// TwinCAT 3 PLC project program1
// ProgramVersion: 3.1.4023.0
// libraries:
//   Tc2_Standard, * (Beckhoff Automation GmbH)
//   Tc2_System, * (Beckhoff Automation GmbH)
//   Tc3_Module, * (Beckhoff Automation GmbH)
// project tree:
//   GVLs/ Common_GVL.TcGVL, ST_Siemens_data_inputs.TcDUT, ST_Siemens_data_outputs.TcDUT, ST_Siemens_other_parameters.TcDUT, ST_Siemens_production_data.TcDUT
//   / PlcTask.TcTTO
//   POUs/ FB_TestFunction.TcPOU, MAIN.TcPOU
// real-time tasks:
//   TASK PlcTask: cycle T#10ms, priority 20, ADS port 350
//   TASK Device 1 (OPC UA Virtual)_Task_58: cycle T#40ms, priority 58, ADS port 351
// I/O:
//   DEVICE Device 1 (OPC UA Virtual), AmsNetId 192.168.0.5.2.1
// variable links:
//   program1/program1 Instance <-> Device 1 (OPC UA Virtual)/Client #1/ServerInterfaces.Communication_with_beckhoff.Bottle_Count
//     PlcTask Inputs/TestData.xBottleCount <-> Inputs/Value
//   program1/program1 Instance <-> Device 1 (OPC UA Virtual)/Client #1/ServerInterfaces.Communication_with_beckhoff.Flow_ml_per_sec
//     PlcTask Inputs/TestData.rFlow_in_ml_s <-> Inputs/Value
//   program1/program1 Instance <-> Device 1 (OPC UA Virtual)/Client #1/ServerInterfaces.Communication_with_beckhoff.LiquidA_in_Bottle
//     PlcTask Inputs/TestData.aryLiquidA_in_bottle <-> Inputs/Value
//     PlcTask Inputs/TestData.aryLiquidA_in_bottle[{0..5}] <-> Inputs/Value[{0..5}]  (6 links)
//   program1/program1 Instance <-> Device 1 (OPC UA Virtual)/Client #1/ServerInterfaces.Communication_with_beckhoff.LiquidB_in_Bottle
//     PlcTask Inputs/TestData.aryLiquidB_in_bottle <-> Inputs/Value
//     PlcTask Inputs/TestData.aryLiquidB_in_bottle[{0..5}] <-> Inputs/Value[{0..5}]  (6 links)
//   program1/program1 Instance <-> Device 1 (OPC UA Virtual)/Client #1/ServerInterfaces.Communication_with_beckhoff.T02_Level_in_L
//     PlcTask Inputs/TestData.rT02_Level_in_L <-> Inputs/Value
//   program1/program1 Instance <-> Device 1 (OPC UA Virtual)/Client #1/ServerInterfaces.Communication_with_beckhoff.Total_Liquid_in_Bottle
//     PlcTask Inputs/TestData.aryTotal_Liquid_in_bottle <-> Inputs/Value
//     PlcTask Inputs/TestData.aryTotal_Liquid_in_bottle[{0..5}] <-> Inputs/Value[{0..5}]  (6 links)

CONFIGURATION program1
    RESOURCE PLC ON TwinCAT3
        TASK PlcTask(INTERVAL := T#10ms, PRIORITY := 20);
        PROGRAM MAIN WITH PlcTask : MAIN;
    END_RESOURCE
END_CONFIGURATION

// ---- GVLs/ST_Siemens_data_inputs.TcDUT
TYPE ST_Siemens_data_inputs :
STRUCT
	FIC_B102 : INT;
	LIC_B101 : INT;
	PS1_RFID_Station : BOOL;
	PS2_Filling_Station : BOOL;
	PS3_Quality_Station : BOOL;
	PS4_End_of_Conveyor : BOOL;
	T01_Low_level : BOOL;
	T01_High_level : BOOL;	
END_STRUCT
END_TYPE

// ---- GVLs/ST_Siemens_data_outputs.TcDUT
TYPE ST_Siemens_data_outputs :
STRUCT
	T01_outlet : BOOL;
	T02_outlet : BOOL;
	Outlet_pump_motor : BOOL;
	Conveyor_motor : BOOL;
	T01_inlet : BOOL;
	T02_inlet : BOOL;	
END_STRUCT
END_TYPE

// ---- GVLs/ST_Siemens_other_parameters.TcDUT
TYPE ST_Siemens_other_parameters :
STRUCT
	Liquid_A_filled : BOOL;
	Liquid_B_filled : BOOL;
	Flow_ml_per_sec : REAL;
	LiquidA_in_Bottle_ml : REAL;
	LiquidB_in_Bottle_ml : REAL;
	T02_Level_in_L : REAL;
	T02_High_Level_limit : REAL;
	T02_Low_Level_limit : REAL;		
END_STRUCT
END_TYPE

// ---- GVLs/ST_Siemens_production_data.TcDUT
TYPE ST_Siemens_production_data :
STRUCT
	Total_Liquid_in_Bottle : ARRAY [1..5] OF REAL;
	LiquidA_in_Bottle : ARRAY [1..5] OF REAL;
	LiquidB_in_Bottle : ARRAY [1..5] OF REAL;
	Bottle_count : INT;
END_STRUCT
END_TYPE

// ---- GVLs/Common_GVL.TcGVL
{attribute 'qualified_only'}
VAR_GLOBAL
	// Scanned values from RFID tags
	{attribute 'OPC.UA.DA' := '1'}
	RFID_LiquidA AT %Q* : INT;
	{attribute 'OPC.UA.DA' := '1'}
	RFID_LiquidB AT %Q* : INT;
	{attribute 'OPC.UA.DA' := '1'}
	Alarm_reset  AT %Q* : BOOL;
	
	// Data from the Siemens Slave PLC
	
    {attribute 'OPC.UA.DA' := '1'}
    {attribute 'OPC.UA.DA.StructuredType' := '1'}
	stSiemens_data_inputs AT %I*  : ST_Siemens_data_inputs;
	
    {attribute 'OPC.UA.DA' := '1'}
    {attribute 'OPC.UA.DA.StructuredType' := '1'}
	stSiemens_data_outputs AT %I*  : ST_Siemens_data_Outputs;
	
    {attribute 'OPC.UA.DA' := '1'}
    {attribute 'OPC.UA.DA.StructuredType' := '1'}
	stSiemens_other_parameters AT %I*  : ST_Siemens_other_parameters;
	
    {attribute 'OPC.UA.DA' := '1'}
    {attribute 'OPC.UA.DA.StructuredType' := '1'}
	stSiemens_Siemens_production_data AT %I* : ST_Siemens_production_data;
	
	
END_VAR

// ---- POUs/MAIN.TcPOU
PROGRAM MAIN
VAR
	fbTestFunction : FB_TestFunction;
END_VAR

END_PROGRAM

// ---- POUs/FB_TestFunction.TcPOU
FUNCTION_BLOCK FB_TestFunction
VAR_INPUT
END_VAR
VAR_OUTPUT
END_VAR
VAR
END_VAR

END_FUNCTION_BLOCK
